FUNCTION_BLOCK FB_NOTT_DELAY_LINES
VAR_INPUT
END_VAR
VAR_OUTPUT
END_VAR
VAR
	NDL1:		FB_MOTOR;
	NDL2:		FB_MOTOR;
	NDL3:		FB_MOTOR;
	NDL4:		FB_MOTOR;
	
	ptrDelayLines:	ARRAY [1..4] OF POINTER TO FB_MOTOR;
	// GUI stuff
	guiShutterIndex:	UINT := 1;	// Index for Shutter Engineering GUI
		
END_VAR

NDL1(
	in_bSafe:=, 
	in_bDisableIfUnsafe:=, 
	sName:= 'NDL1', 
	nNOVRAM_DevId:= 6, 
	nNOVRAM_Offset:= 1000);
	
NDL2(
	in_bSafe:=, 
	in_bDisableIfUnsafe:=, 
	sName:= 'NDL2', 
	nNOVRAM_DevId:= 6, 
	nNOVRAM_Offset:= 2000);
	
NDL3(
	in_bSafe:=, 
	in_bDisableIfUnsafe:=, 
	sName:= 'NDL3', 
	nNOVRAM_DevId:= 6, 
	nNOVRAM_Offset:= 3000);
	
NDL4(
	in_bSafe:=, 
	in_bDisableIfUnsafe:=, 
	sName:= 'NDL4', 
	nNOVRAM_DevId:= 6, 
	nNOVRAM_Offset:= 4000);
	

M_Configure();

METHOD M_Configure : BOOL
VAR_INPUT
END_VAR

ptrDelayLines[1] := ADR(NDL1);
ptrDelayLines[2] := ADR(NDL2);
ptrDelayLines[3] := ADR(NDL3);
ptrDelayLines[4] := ADR(NDL4);
END_METHOD

END_FUNCTION_BLOCK

(* stored: Version 1.1.0.1, ProductVersion 3.1.4024.12
   POU FB_NOTT_DELAY_LINES: Id {775cfb6f-4389-4959-8f2c-a4b0ad5c5054}, SpecialFunc None
   Method M_Configure: Id {fce285f8-42af-45ec-adbe-2e2f465358d7} *)
